(****************************************************************************************)
(*							Beckhoff Automation Poland									*)
(*								F_MaskWord v1.0											*)
(*									15.02.2010											*)
(*		Funkcja wyciagajaca  okreslona ilosc Bitow ze ze zmiennej typu WORD				*)
(*							 wyjscie typu WORD											*)
(*______________________________________________________________________________________*)
FUNCTION F_MaskWord : WORD
VAR_INPUT
	wIn	:	WORD; (*Wejscie*)
	wNo	:	WORD; (*Ilosc bitow, zaczynajac od LSB*)
END_VAR

CASE wNo OF
	0:
	F_MaskWord := wIn AND 2#0;
	1:
	F_MaskWord := wIn AND 2#1;
	2:
	F_MaskWord := wIn AND 2#11;
	3:
	F_MaskWord := wIn AND 2#111;
	4:
	F_MaskWord := wIn AND 2#1111;
	5:
	F_MaskWord := wIn AND 2#11111;
	6:
	F_MaskWord := wIn AND 2#111111;
	7:
	F_MaskWord := wIn AND 2#1111111;
	8:
	F_MaskWord := wIn AND 2#11111111;
	9:
	F_MaskWord := wIn AND 2#111111111;
	10:
	F_MaskWord := wIn AND 2#1111111111;
	11:
	F_MaskWord := wIn AND 2#11111111111;
	12:
	F_MaskWord := wIn AND 2#111111111111;
	13:
	F_MaskWord := wIn AND 2#1111111111111;
	14:
	F_MaskWord := wIn AND 2#11111111111111;
	15:
	F_MaskWord := wIn AND 2#111111111111111;
	16:
	F_MaskWord := wIn;
END_CASE

END_FUNCTION

(* stored: Version 1.1.0.1, ProductVersion 3.1.4026.13, FileIdentifier a915b286a74137693d9fcdee9515a9a301544241, FileSignature 14cefa980327706f442688fcdf2041dd304d4f97550828ea500a3e308750ee524a558e40ec796fb8522f4c7e7ea446424c7d46938b1496454ad5614b3869e80a335c21ac54767de0cae84ff3518d4df61a75d4a093dce5af1b9519707224d67620fe8ba73f9d50c3a55964f58240e42c225e6ece2bfa3ffd17e91cebafc94b39b1f797bb4f3828f3a390c5edd512b6feb035ad8ed49adaff4e96232c1c3905240cd9de61bb7a58b6f7b7df6f7a2b5a2299cbf237c51599c8d1d87ebacbc69a7ed1c5c57ef7f960f19d0f7c490e7704fb13e2d9fbb5cd0ea952e3c191f0a0cd271c1376037bcd3d3bfda7bd5d67662d0096ee56845b1402c30a029321d8982b40
   POU F_MaskWord: Id {968f3ca7-c1c8-4d7e-bb4e-50e46c45be6c}, SpecialFunc None *)
